// TIA Portal project "project" (V15.1)
// Vorlageprojekt für das Buch mit Zielsystem S7-1200

(* hardware
DEVICE "S7-1200-Station_1"  S7-1200 Station
   slot 0: "Baugruppenträger_0"  Rack  V1.0
   slot 1: "PLC_1"  CPU 1211C DC/DC/DC  6ES7 211-1AE40-0XB0  V4.1
*)

// ===== PLC "PLC_1"  CPU 1211C DC/DC/DC =====

VAR_GLOBAL   // PLC tag table "Standard-Variablentabelle"
   "Entry convenyor" AT %A0.0 : Bool;
   "Tag_2" AT %E0.0 : Bool;
   "start" AT %E0.1 : Bool;
   "Reset Light" AT %Q1.2 : Bool;
   "Stop Light" AT %Q1.3 : Bool;
   "Exit convenyor" AT %Q0.2 : Bool;
   "Stop Blade" AT %Q0.1 : Bool;
   "Start Light" AT %Q1.1 : Bool;
   "sensor vision" AT %ID30 : DWord;
   "Tag_10" AT %Q1.4 : Bool;
   "Tag_11" AT %Q0.3 : Bool;
   "Tag_12" AT %QD30 : DWord;
   "Tag_13" AT %Q1.5 : Bool;
   "Tag_14" AT %Q0.5 : Bool;
   "Tag_15" AT %Q1.6 : Bool;
   "Tag_16" AT %Q0.7 : Bool;
   "stop" AT %I1.3 : Bool;
   "Tag_1" AT %I1.2 : Bool;
   "timmer 1 valve" AT %Q1.4 : Bool;
   "sorter 1 turn" AT %Q0.3 : Bool;
   "sorter 1 turn(1)" AT %Q0.3 : Bool;
   "timmer 2 valve" AT %Q1.5 : Bool;
   "sorter 2 turn" AT %Q0.5 : Bool;
   "timmer 3 valve" AT %Q1.6 : Bool;
   "sorting 3 turn" AT %Q0.7 : Bool;
   "Tag_3" AT %I0.3 : Bool;
   "sorter 1 belt" AT %Q0.4 : Bool;
   "sorter 2 belt" AT %Q0.6 : Bool;
   "sorter 3 belt" AT %Q1.0 : Bool;
END_VAR

// folder: System blocks/Program resources

DATA_BLOCK "IEC_Timer_0_DB"   // DB1
{ S7_Optimized_Access := 'TRUE' }
AUTHOR : Simatic
FAMILY : IEC
NAME : IEC_TMR
VERSION : 1.0
// stored: InstanceOfName IEC_TIMER
"IEC_TIMER"
BEGIN
END_DATA_BLOCK

DATA_BLOCK "IEC_Timer_0_DB_1"   // DB2
{ S7_Optimized_Access := 'TRUE' }
AUTHOR : Simatic
FAMILY : IEC
NAME : IEC_TMR
VERSION : 1.0
// stored: InstanceOfName IEC_TIMER
"IEC_TIMER"
BEGIN
END_DATA_BLOCK

DATA_BLOCK "timer 4"   // DB3
{ S7_Optimized_Access := 'TRUE' }
AUTHOR : Simatic
FAMILY : IEC
NAME : IEC_TMR
VERSION : 1.0
// stored: InstanceOfName IEC_TIMER
"IEC_TIMER"
BEGIN
END_DATA_BLOCK

DATA_BLOCK "timer 2"   // DB4
{ S7_Optimized_Access := 'TRUE' }
AUTHOR : Simatic
FAMILY : IEC
NAME : IEC_TMR
VERSION : 1.0
// stored: InstanceOfName IEC_TIMER
"IEC_TIMER"
BEGIN
END_DATA_BLOCK

DATA_BLOCK "timer 3"   // DB6
{ S7_Optimized_Access := 'TRUE' }
AUTHOR : Simatic
FAMILY : IEC
NAME : IEC_TMR
VERSION : 1.0
// stored: InstanceOfName IEC_TIMER
"IEC_TIMER"
BEGIN
END_DATA_BLOCK

// folder: (top level)

FUNCTION "MHJ-PLC-Lab-Function-S71200" : Void   // FC9000, SCL
{ S7_Optimized_Access := 'TRUE' }
VERSION : 0.1
   VAR_TEMP
      rdTimeReturn : Int;
      outputTime : DTL;
      SyncVal : Byte;
      forVal : Int;
      forVal_2 : Int;
      Value : Byte;
   END_VAR
   VAR CONSTANT
      CompVal : Byte := 16#34;
      Value_01 : Byte := 16#11;
      Value_01_DW : DWord := 16#A165_D992;
      Value_02_DW : DWord := 16#58BE_4401;
   END_VAR
BEGIN

   #Value:=PEEK(area := 16#82,
        dbNumber := 0,
        byteOffset := 511);
   #Value := #Value + 1;

   POKE(area := 16#82,
        dbNumber := 0,
        byteOffset := 511,
        value := #Value);

   POKE(area:=16#81,
        dbNumber:=0,
        byteOffset:=1016,
        value:=#Value_01_DW);
   POKE(area := 16#81,
        dbNumber := 0,
        byteOffset := 1020,
        value := #Value_02_DW);

   POKE(area := 16#81,
        dbNumber := 0,
        byteOffset := 511,
        value := B#16#00);

   FOR #forVal := 0 TO 120 DO
       FOR #forVal_2:=0 TO 10 DO
           #rdTimeReturn:=RD_SYS_T(#outputTime);
           #rdTimeReturn := WR_SYS_T(#outputTime);
           #rdTimeReturn := RD_SYS_T(#outputTime);
           #rdTimeReturn := WR_SYS_T(#outputTime);
       END_FOR;
       #SyncVal:= PEEK(area := 16#81,
                      dbNumber := 0,
                      byteOffset := 511);
       IF #SyncVal = #CompVal THEN
          GOTO M_1;
       END_IF;
   END_FOR;
   RETURN;

   M_1:
   POKE(area := 16#81,
        dbNumber := 0,
        byteOffset := 511,
        value := B#16#0);
END_FUNCTION

ORGANIZATION_BLOCK "Main"   // OB1, LAD, ProgramCycle
TITLE = "Main Program Sweep (Cycle)"
{ S7_Optimized_Access := 'TRUE' }
VERSION : 0.1
   VAR_INPUT
      Initial_Call : Bool;   // Initial call of this OB
      Remanence : Bool;   // =True, if remanent data are available
   END_VAR
   VAR CONSTANT
      start : Bool;
   END_VAR
BEGIN

REGION Network 1: Konnektierungsbaustein für PLC-Lab
   // Im Netzwerk 1 wird der Konnektierungsbaustein für PLC-Lab aufgerufen.
   // Dieser Aufruf darf nicht entfernt werden!
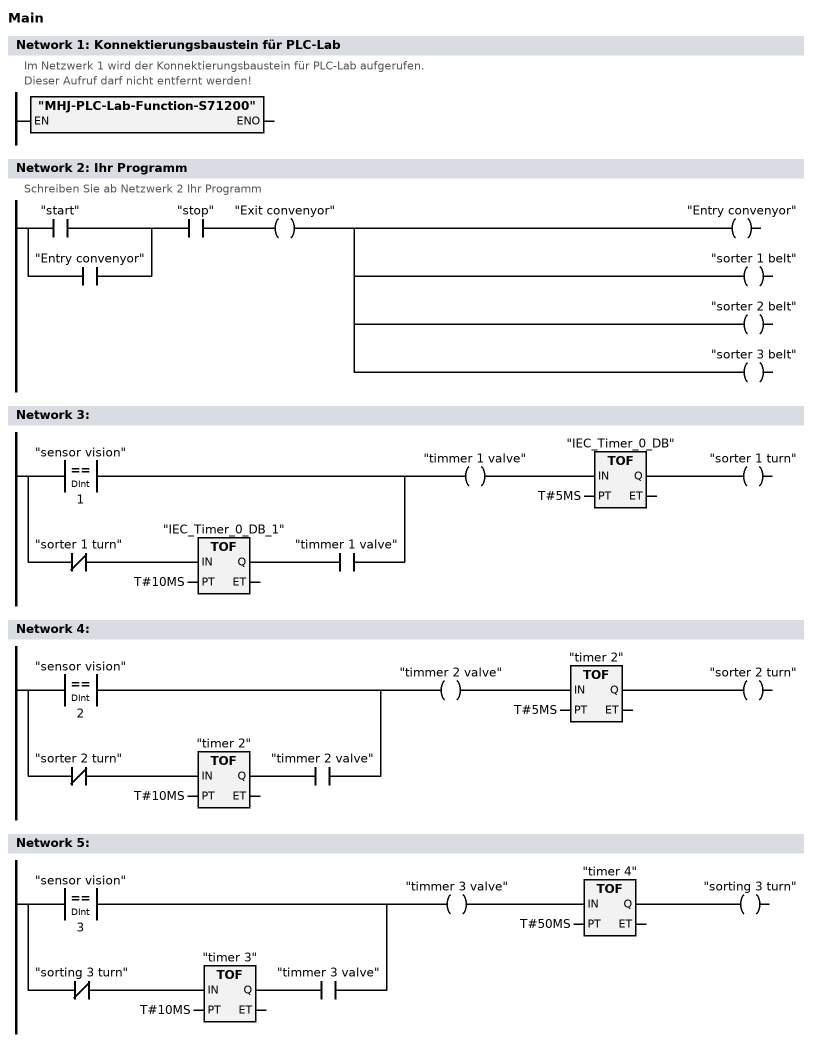
   RUNG wire#powerrail
      "MHJ-PLC-Lab-Function-S71200"()
   END_RUNG
   // the same network as SCL:
   "MHJ-PLC-Lab-Function-S71200"();
END_REGION

REGION Network 2: Ihr Programm
   // Schreiben Sie ab Netzwerk 2 Ihr Programm
   RUNG wire#powerrail
      Contact( "start" )
      wire#w1
      Contact( "stop" )
      Coil( "Exit convenyor" )
      wire#w2
      Coil( "Entry convenyor" )
   END_RUNG
   RUNG wire#powerrail
      Contact( "Entry convenyor" )
   END_RUNG wire#w1
   RUNG wire#w2
      Coil( "sorter 1 belt" )
   END_RUNG
   RUNG wire#w2
      Coil( "sorter 2 belt" )
   END_RUNG
   RUNG wire#w2
      Coil( "sorter 3 belt" )
   END_RUNG
   // the same network as SCL:
   "Exit convenyor" := ("start" OR "Entry convenyor") AND "stop";
   "Entry convenyor" := "Exit convenyor";
   "sorter 1 belt" := "Exit convenyor";
   "sorter 2 belt" := "Exit convenyor";
   "sorter 3 belt" := "Exit convenyor";
END_REGION

REGION Network 3
   "IEC_Timer_0_DB_1".TOF(IN := NOT "sorter 1 turn", PT := T#10MS);
   "timmer 1 valve" := ("sensor vision" = 1) OR ("IEC_Timer_0_DB_1".Q AND "timmer 1 valve");
   "IEC_Timer_0_DB".TOF(IN := "timmer 1 valve", PT := T#5MS);
   "sorter 1 turn" := "IEC_Timer_0_DB".Q;
END_REGION

REGION Network 4
   "timer 2".TOF(IN := NOT "sorter 2 turn", PT := T#10MS);
   "timmer 2 valve" := ("sensor vision" = 2) OR ("timer 2".Q AND "timmer 2 valve");
   "timer 2".TOF(IN := "timmer 2 valve", PT := T#5MS);
   "sorter 2 turn" := "timer 2".Q;
END_REGION

REGION Network 5
   "timer 3".TOF(IN := NOT "sorting 3 turn", PT := T#10MS);
   "timmer 3 valve" := ("sensor vision" = 3) OR ("timer 3".Q AND "timmer 3 valve");
   "timer 4".TOF(IN := "timmer 3 valve", PT := T#50MS);
   "sorting 3 turn" := "timer 4".Q;
END_REGION
END_ORGANIZATION_BLOCK